(* CoDeSys 2.3 export: ETAGE_RDC.EXP *)

(* POU Initialisation_Standby/ETAGE_RDC, SFC *)
PROGRAM ETAGE_RDC
VAR
END_VAR
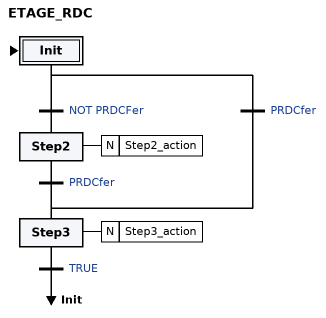
INITIAL_STEP Init:
END_STEP
TRANSITION FROM Init TO Step2 := NOT PRDCFer;
END_TRANSITION
TRANSITION FROM Init TO Step3 := PRDCfer;
END_TRANSITION
STEP Step2:
	Step2_action(N);
END_STEP
TRANSITION FROM Step2 TO Step3 := PRDCfer;
END_TRANSITION
STEP Step3:
	Step3_action(N);
END_STEP
TRANSITION FROM Step3 TO Init := TRUE;
END_TRANSITION

ACTION Step2_action:
FRDC:=TRUE;
END_ACTION

ACTION Step3_action:
FRDC:=FALSE;
Quel_Etage();
END_ACTION
END_PROGRAM
